// TIA Portal V16 export
// export: Created 2021-08-30T13:41:01.928247Z, ExportSetting WithDefaults, DisplayName Totally Integrated Automation Portal, DisplayVersion V16 Update 3, DisplayName TIA Portal Version Control Interface, DisplayVersion V16 Update 2, DisplayName TIA Portal Openness, DisplayVersion V16 Update 3, DisplayName TIA Portal Teamcenter Gateway, DisplayVersion V16, DisplayName STEP 7 Professional, DisplayVersion V16 Update 3, DisplayName STEP 7 Safety, DisplayVersion V16, DisplayName WinCC Advanced, DisplayVersion V16 Update 3
DATA_BLOCK "dtPropDpump"   // DB14
{ S7_Optimized_Access := 'TRUE' }
VERSION : 0.1
// stored: AutoNumber true, DBAccessibleFromOPCUA true, IsOnlyStoredInLoadMemory false, IsRetainMemResEnabled false, IsWriteProtectedInAS false, MemoryReserve 100
   VAR
      dp101 : "PropDosing";
      dp501 : "PropDosing";
      dp502 : "PropDosing";
      dp801 : "PropDosing";
      dp802 : "PropDosing";
      dp803 : "PropDosing";
      dp1001 : "PropDosing";
   END_VAR
BEGIN
END_DATA_BLOCK
